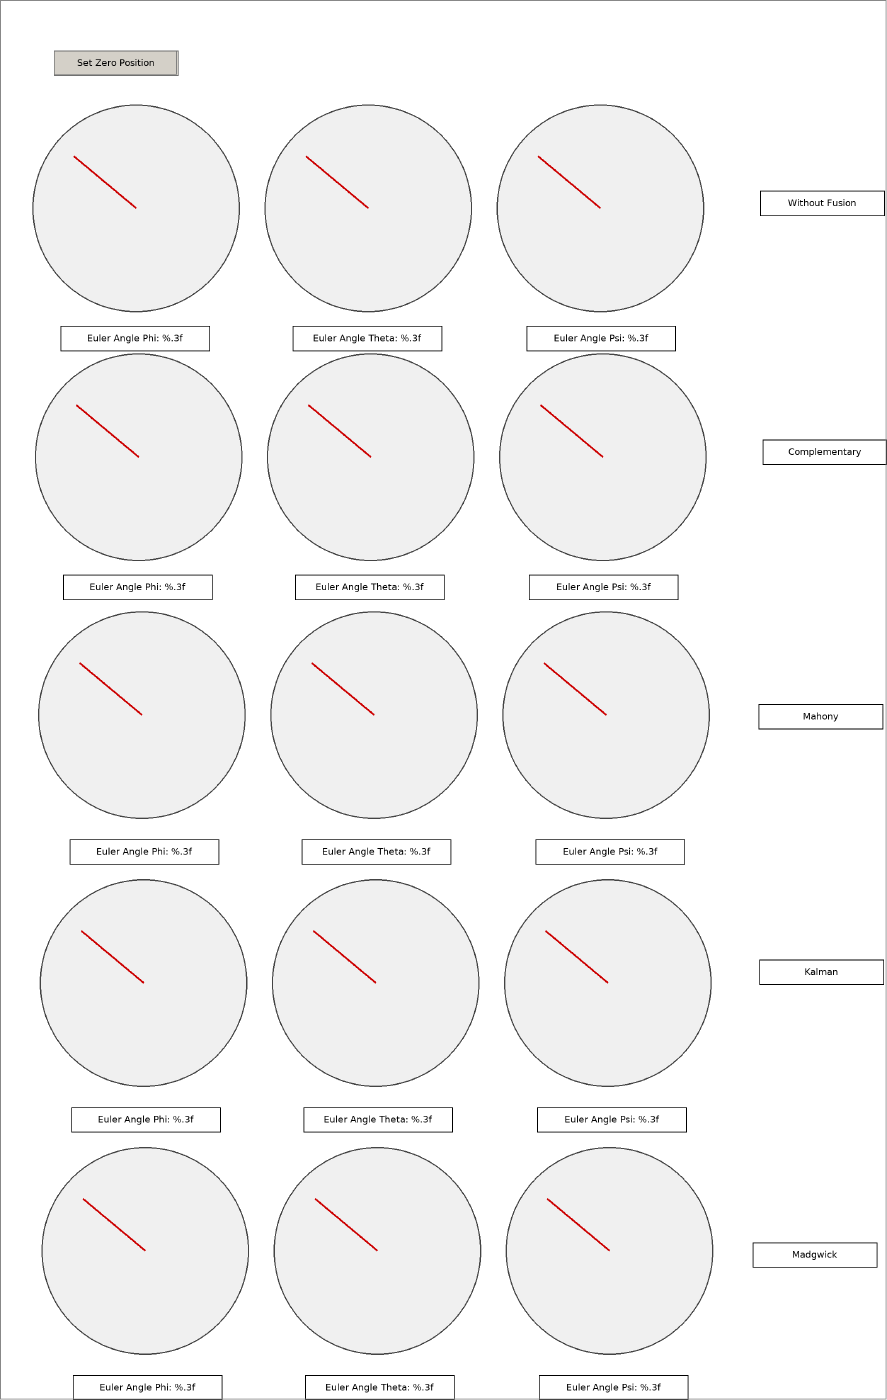
VISUALIZATION Visualization_all  // 1070x1688
    Button (65,61 150x30), "Set Zero Position", colour toggle: MAIN.bReady
        p2175578022: 16#FF808080
        p573394764: 16#FF80FF80
        tap MAIN.bReset
    Meter360 (42,426 250x250), value: MAIN.fbComplementaryFilter.stEulerAngle_deg.X, style: Meter-Meter360-Gray, scale format: %d, scale -180..180
        p518627256: °
    Meter360 (322,426 250x250), value: MAIN.fbComplementaryFilter.stEulerAngle_deg.Y, style: Meter-Meter360-Gray, scale format: %d, scale -180..180
        p518627256: °
    Meter360 (602,426 250x250), value: MAIN.fbComplementaryFilter.stEulerAngle_deg.Z, style: Meter-Meter360-Gray, scale format: %d, scale -180..180
        p518627256: °
    Rectangle (76,693 180x30), "Euler Angle Phi: %.3f", text variable: MAIN.fbComplementaryFilter.stEulerAngle_deg.X
    Rectangle (356,693 180x30), "Euler Angle Theta: %.3f", text variable: MAIN.fbComplementaryFilter.stEulerAngle_deg.Y
    Rectangle (638,693 180x30), "Euler Angle Psi: %.3f", text variable: MAIN.fbComplementaryFilter.stEulerAngle_deg.Z
    Meter360 (46,737 250x250), value: MAIN.fbMahonyFilter.stEulerAngle_deg.X, style: Meter-Meter360-Gray, scale format: %d, scale -180..180
        p518627256: °
    Meter360 (326,737 250x250), value: MAIN.fbMahonyFilter.stEulerAngle_deg.Y, style: Meter-Meter360-Gray, scale format: %d, scale -180..180
        p518627256: °
    Meter360 (606,737 250x250), value: MAIN.fbMahonyFilter.stEulerAngle_deg.Z, style: Meter-Meter360-Gray, scale format: %d, scale -180..180
        p518627256: °
    Rectangle (84,1012 180x30), "Euler Angle Phi: %.3f", text variable: MAIN.fbMahonyFilter.stEulerAngle_deg.X
    Rectangle (364,1012 180x30), "Euler Angle Theta: %.3f", text variable: MAIN.fbMahonyFilter.stEulerAngle_deg.Y
    Rectangle (646,1012 180x30), "Euler Angle Psi: %.3f", text variable: MAIN.fbMahonyFilter.stEulerAngle_deg.Z
    Meter360 (48,1060 250x250), value: MAIN.fbKalmanFilter.stEulerAngle_deg.X, style: Meter-Meter360-Gray, scale format: %d, scale -180..180
        p518627256: °
    Meter360 (328,1060 250x250), value: MAIN.fbKalmanFilter.stEulerAngle_deg.Y, style: Meter-Meter360-Gray, scale format: %d, scale -180..180
        p518627256: °
    Meter360 (608,1060 250x250), value: MAIN.fbKalmanFilter.stEulerAngle_deg.Z, style: Meter-Meter360-Gray, scale format: %d, scale -180..180
        p518627256: °
    Rectangle (86,1335 180x30), "Euler Angle Phi: %.3f", text variable: MAIN.fbKalmanFilter.stEulerAngle_deg.X
    Rectangle (366,1335 180x30), "Euler Angle Theta: %.3f", text variable: MAIN.fbKalmanFilter.stEulerAngle_deg.Y
    Rectangle (648,1335 180x30), "Euler Angle Psi: %.3f", text variable: MAIN.fbKalmanFilter.stEulerAngle_deg.Z
    Meter360 (50,1383 250x250), value: MAIN.fbMadgwickFilter.stEulerAngle_deg.X, style: Meter-Meter360-Gray, scale format: %d, scale -180..180
        p518627256: °
    Meter360 (330,1383 250x250), value: MAIN.fbMadgwickFilter.stEulerAngle_deg.Y, style: Meter-Meter360-Gray, scale format: %d, scale -180..180
        p518627256: °
    Meter360 (610,1383 250x250), value: MAIN.fbMadgwickFilter.stEulerAngle_deg.Z, style: Meter-Meter360-Gray, scale format: %d, scale -180..180
        p518627256: °
    Rectangle (88,1658 180x30), "Euler Angle Phi: %.3f", text variable: MAIN.fbMadgwickFilter.stEulerAngle_deg.X
    Rectangle (368,1658 180x30), "Euler Angle Theta: %.3f", text variable: MAIN.fbMadgwickFilter.stEulerAngle_deg.Y
    Rectangle (650,1658 180x30), "Euler Angle Psi: %.3f", text variable: MAIN.fbMadgwickFilter.stEulerAngle_deg.Z
    RoundedRectangle (920,530 150x30), "Complementary"
    RoundedRectangle (915,849 150x30), "Mahony"
    RoundedRectangle (916,1157 150x30), "Kalman"
    RoundedRectangle (908,1498 150x30), "Madgwick"
    Meter360 (39,126 250x250), value: MAIN.stEulerAngle_Gyro.X, style: Meter-Meter360-Gray, scale format: %d, scale -180..180
        p518627256: °
    Meter360 (319,126 250x250), value: MAIN.stEulerAngle_Gyro.Y, style: Meter-Meter360-Gray, scale format: %d, scale -180..180
        p518627256: °
    Meter360 (599,126 250x250), value: MAIN.stEulerAngle_Gyro.Z, style: Meter-Meter360-Gray, scale format: %d, scale -180..180
        p518627256: °
    Rectangle (73,393 180x30), "Euler Angle Phi: %.3f", text variable: MAIN.stEulerAngle_Gyro.X
    Rectangle (353,393 180x30), "Euler Angle Theta: %.3f", text variable: MAIN.stEulerAngle_Gyro.Y
    Rectangle (635,393 180x30), "Euler Angle Psi: %.3f", text variable: MAIN.stEulerAngle_Gyro.Z
    RoundedRectangle (917,230 150x30), "Without Fusion"
END_VISUALIZATION

(* stored: Version 1.1.0.1, ProductVersion 3.1.4024.13
   Visu Visualization_all: Id {fe0bd2ba-2d98-4aa7-9765-eb93a10851ca} *)
